// TIA Portal V19 export
FUNCTION "HambaFiller" : Void   // FC100, STL
TITLE = Hamba Filler
{ S7_Optimized_Access := 'TRUE' }
VERSION : 0.0
// Comment
// stored: AutoNumber false
BEGIN

NETWORK
TITLE = CIP of Transfer line
      CLR;

      A     "CIP_Hamba_bit_00";
      JC    M015;

      A     "CIP_Hamba_bit_02";  // If system is requested to stop
      AN    "CIP_Route_Request";  // by loss of Route request
      JC    M015;  // It does a controlled shutdown

      A     "CIP_Hamba_bit_02";  // Once CIP Route is started it continues
      JC    M002;  // Unless the Route request is lost


      A     "CIP_Route_Request";
      AN    "Product_Request";
      AN    "Steam_Request";
      A     "CIP Stop Push Button";
      AN    "RTE_404_DB".HMI.RUNNING;
      JCN   M001;

      S     "CIP_Hamba_bit_02";
M002: R     "MY0902";  //turn off steam supply
      R     "MY0909";  //turn off steam to barrier
      A     "CIP_Hamba_bit_03";  //Once Y0909R is proved stop checking
      JC    M016;

      A     "Y0909R";  //check valve de-energised
      A     "PG_Devices".DI_100_005_X06_X1_3p2;  // Polygon Filler transfer line blanked off
      JCN   M001;

      S     "CIP_Hamba_bit_03";
M016: S     "MY0908";  //open 'product' route
      S     "MY0910";  //open 'product' route

      A     "Y0908S";  //check valve energised
      A     "Y0910S";  //check valve energised
      JCN   M001;

      S     "M_Cip_Route";
      S     "CIP_Hamba_bit_00";
      JU    M001;

// Start of Loss of CIP Route Request shutdown sequence
M015: CLR;
      A     "CIP_Hamba_bit_01";  //Awaiting CIP Drain Timer End
      JC    M013;

      A     "CIP_Route_Request";
      A     "CIP Stop Push Button";
      S     "M_Cip_Route";  //CORRECT?

      A     "CIP_Route_Request";
      AN    "CIP_Hamba_bit_04";  // Once Shutdown has started
      JC    M001;  // It continues until completed

      S     "CIP_Hamba_bit_04";
      R     "MY0910";
      R     "M_Cip_Route";
      A     "CIP_Hamba_bit_05";  //Once Y0910R is proved stop checking
      JC    M014;

      A     "Y0910R";  //check valve de-energised
      JCN   M001;

      S     "CIP_Hamba_bit_05";
M014: S     "MY0911";
      A     "Y0911S";  //check valve energised
      JCN   M001;

      S     "TIM57";  // DrainingHambaTime
      S     "CIP_Hamba_bit_01";
      JU    M001;

M013: CLR;
      A     "Tag_69";
      JC    M001;
      R     "MY0911";
      R     "MY0908";
      R     "CIP_Hamba_bit_00";
      R     "CIP_Hamba_bit_01";
      R     "CIP_Hamba_bit_02";
      R     "CIP_Hamba_bit_03";
      R     "CIP_Hamba_bit_04";
      R     "CIP_Hamba_bit_05";

M001: CLR;
      A     "CIP_Running";
      =     "MX0913";  //set cip running bit

      A     "M_Cip_Route";  //cip route is active
      A(;
      O     "ItemAlarmsOP".Item[20];  //FB_FAULT_VALVE_09_05
      O     "ItemAlarmsOP".Item[23];  //FB_FAULT_VALVE_09_08
      O     "ItemAlarmsOP".Item[24];  //FB_FAULT_VALVE_09_09
      O     "ItemAlarmsOP".Item[25];  //FB_FAULT_VALVE_09_10
      O     "ItemAlarmsOP".Item[26];  //FB_FAULT_VALVE_09_11
      ON    "PG_Devices".DI_100_005_X06_X1_3p2;  // Polygon Filler transfer line blanked off
      );
      R     "M_Cip_Route";  //reset cip route active flag if valve in fault

NETWORK
TITLE = CIp Stop Push Button Operated Alarm and Stop CIP route signal
      AN    "CIP Stop Push Button";
      S     "ProcessAndPbAlarms"."A"[63];  //A63_Stop_CIP_PB_Operated
      R     "M_Cip_Route";

NETWORK
TITLE = SIP of Transfer line
      A     "steam_lp_request";  // If LP steam is requested
      R     "MY0903";  //
      S     "MY0902";

      A     "steam_lp_request";  // If LP steam is requested
      AN    "MY0903";  // if Y0903 is being asked to close
      A     "MY0902";  // and Y0902 is being asked to open
      =     "M_LP_Steam_ON";  // then, inform that the LP steam request has been actioned


      CLR;

      A     "SIP_Hamba_bit_00";
      JC    M005;

      A     "SIP_Hamba_bit_02";  // If system is requested to stop
      A(;  // After it has been started
      ON    "Steam_Request";  // It does a controlled shutdown
      ON    "Barrier_Sterile";
      );
      S     "SIP_Hamba_bit_00";
      JC    M005;

      A     "Steam_Request";
      A     "Barrier_Sterile";
      JCN   M004;

      S     "SIP_Hamba_bit_02";
      R     "MY0902";
      R     "MY0910";
      R     "MY0911";
      A     "SIP_Hamba_bit_04";  //Once Y0910R and Y0911R are proved
      JC    M003;  //Stop checking

      A     "Y0910R";  //check valve de-energised
      A     "Y0911R";  //check valve de-energised
      JCN   M004;

      S     "SIP_Hamba_bit_04";
M003: S     "MY0908";
      S     "MY0909";
      A     "Y0908S";  //check valve energised
      A     "Y0909S";  //check valve energised
      JCN   M004;

      S     "MY0903";
      S     "M_Sip_Steam";
      S     "SIP_Hamba_High_SteamPres";
      R     "SIP_Hamba_Low_SteamPres";
      S     "SIP_Hamba_bit_00";
      JU    M004;

// Start of Loss of SIP Route Request shutdown sequence
M005: CLR;
      A     "SIP_Hamba_bit_01";
      JC    M017;

      A     "Steam_Request";
      AN    "SIP_Hamba_bit_03";
      JC    M004;

      S     "SIP_Hamba_bit_03";
      R     "MY0908";
      R     "SIP_Hamba_High_SteamPres";
      A     "Y0908R";  //check valve de-energised
      JCN   M004;

      R     "M_Sip_Steam";
      R     "MY0903";
      S     "MY0902";
      S     "SIP_Hamba_Low_SteamPres";
      S     "SIP_Hamba_bit_01";
      JC    M004;

M017: CLR;
      A     "ATI";
      R     "SIP_Hamba_bit_00";
      R     "SIP_Hamba_bit_01";
      R     "SIP_Hamba_bit_02";
      R     "SIP_Hamba_bit_03";
      R     "SIP_Hamba_bit_04";
      R     "SIP_Hamba_bit_05";

M004: NOP   0;

      AN    "Barrier_Sterile";
      R     "SIP_Hamba_High_SteamPres";
      R     "SIP_Hamba_Low_SteamPres";
      CLR;

      A(;
      O     "ItemAlarmsOP".Item[23];  //FB_FAULT_VALVE_09_08
      O     "ItemAlarmsOP".Item[24];  //FB_FAULT_VALVE_09_09
      O     "ItemAlarmsOP".Item[25];  //FB_FAULT_VALVE_09_10
      O     "ItemAlarmsOP".Item[26];  //FB_FAULT_VALVE_09_11
      O     "steam_lp_request";  // If LP steam is requested
      );
      R     "M_Sip_Steam";
      CLR;

      AN    "ItemAlarmsOP".Item[23];  //FB_FAULT_VALVE_09_08
      AN    "ItemAlarmsOP".Item[24];  //FB_FAULT_VALVE_09_09
      AN    "ItemAlarmsOP".Item[25];  //FB_FAULT_VALVE_09_10
      AN    "ItemAlarmsOP".Item[26];  //FB_FAULT_VALVE_09_11
      A     "MY0903";
      S     "M_Sip_Steam";
      CLR;

      AN    "TANK STERILE";
      R     "M_Barrier_Sterile";
      CLR;
      A     "Y0119S";
      R     "MY0902";
      R     "MY0903";
      R     "MY0909";
      R     "SIP_Hamba_Low_SteamPres";

NETWORK
TITLE = SIP of Transfer line Temp. check/alarm high
      A     "MY0903";
      A(;
      L     "MeasuredValues".TT0950REAL;
      L     "Setpoints_Hamba".TT0950BarrierTempHigh;
      <R;
      );
      L     "TIMER DATA BLOCK".SETPOINT_TIMER_58;
      SD    "Tag_99";
      NOP   0;
      NOP   0;
      NOP   0;
      A     "Tag_99";
      S     "ProcessAndPbAlarms"."A"[59];  //A59_TT0950TooLow
      R     "M_Sip_Steam";

NETWORK
TITLE = SIP of Transfer line Temp. check/alarm low
      A     "MY0902";
      A(;
      L     "MeasuredValues".TT0950REAL;
      L     "Setpoints_Hamba".TT0950BarrierTempLow;
      <R;
      );
      L     "TIMER DATA BLOCK".SETPOINT_TIMER_59;
      SD    "Tag_100";
      NOP   0;
      NOP   0;
      NOP   0;
      A     "Tag_100";
      S     "ProcessAndPbAlarms"."A"[60];  //A60_TT0950Low

NETWORK
TITLE = Product Routing
// ; Product available
      A     "M_PROD_AVAILABLE";
      FP    "One_shut_on";
      S     "M_Product_Available";

      AN    "M_PROD_AVAILABLE";
      FP    "One_shut_off";
      R     "M_Product_Available";

//; Product Routing

      A     "Prod_Hamba_bit_00";
      JC    M006;

      A     "Prod_Hamba_bit_08";  //If Product Route request
      AN    "Product_Request";  //Started but not complete
      S     "Prod_Hamba_bit_00";  //When Product request lost
      JC    M006;  //Go to Prod Route Shutdown

      A     "Product_Request";
      A     "MY0902";  //Cross check. V0902 will be energised if route selected.
      JCN   M007;
      S     "Prod_Hamba_bit_08";
      R     "MY0906";
      R     "MY0907";
      R     "MY0912";

      A     "Prod_Hamba_bit_09";  //Jump if Y0906R, Y0907R
      JC    M012;  //& Y0912R have been proved

      A     "Y0906R";  //check valve de-energised
      A     "Y0907R";  //check valve de-energised
      A     "Y0912R";  //check valve de-energised
      A     "Y0908R";  //check valve de-energised, closed on loss of "Steam_Request" Network 3
      JCN   M007;

      S     "Prod_Hamba_bit_09";
M012: S     "MY0904";
      S     "MY0905";
      A     "Y0904S";  //check valve energised
      A     "Y0905S";  //check valve energised
      JCN   M007;

      S     "M_Product_Route";
      S     "Prod_Hamba_bit_00";
      JU    M007;

//Start of loss of Product Route signal
M006: CLR;
      A     "Prod_Hamba_bit_01";
      JC    M00c;

      A     "Product_Request";  //Once Poduct route Shutdown
      AN    "Prod_Hamba_bit_10";  //Started set to ensure finishes
      JC    M007;

      S     "Prod_Hamba_bit_10";
      R     "M_Product_Route";
      R     "MY0904";
      R     "MY0905";
      S     "DisableMonitoringTT0951";
      A     "Prod_Hamba_bit_11";  //Jump if Y0904R & Y0905R
      JC    M008;  //have been proved

      A     "Y0904R";  //check valve de-energised
      A     "Y0905R";  //check valve de-energised
      JCN   M007;

      S     "Prod_Hamba_bit_11";
M008: S     "MY0907";
      S     "MY0912";
      A     "Prod_Hamba_bit_12";  //Jump if Y0907S & Y0912S
      JC    M009;  //have been proved

      A     "Y0907S";  //check valve energised
      A     "Y0912S";  //check valve energised
      JCN   M007;

      S     "Prod_Hamba_bit_12";
M009: S     "MY0906";
      A     "Y0906S";  //check valve energised
      JCN   M007;

      S     "TIM63";  // Y0912PurgeBarrierTime
      S     "Prod_Hamba_bit_01";
      JU    M007;

M00c: CLR;
      A     "Prod_Hamba_bit_02";
      JC    M00d;

      A     "Tag_71";
      JC    M007;
      R     "MY0912";
      R     "DisableMonitoringTT0951";
      A     "Y0912R";  //check valve de-energised
      JCN   M007;

      S     "Prod_Hamba_bit_02";
      JU    M007;

M00d: CLR;
      A     "ATI";
      R     "Prod_Hamba_bit_00";
      R     "Prod_Hamba_bit_01";
      R     "Prod_Hamba_bit_02";
      R     "Prod_Hamba_bit_08";
      R     "Prod_Hamba_bit_09";
      R     "Prod_Hamba_bit_10";
      R     "Prod_Hamba_bit_11";
      R     "Prod_Hamba_bit_12";

M007: CLR;
      AN    "Product_Request";
      R     "Prod_Hamba_bit_03";
      R     "Prod_Hamba_bit_04";
      R     "Prod_Hamba_bit_05";
      R     "Prod_Hamba_bit_06";
      R     "ProcessAndPbAlarms"."A"[61];  //A61_Hamba_Valve_Fault
      R     "ProcessAndPbAlarms"."A"[62];  //A62_Hamba_Barrier_low
      BEC;

//; Valve FB-error

      A     "Prod_Hamba_bit_03";
      AN    "Prod_Hamba_bit_04";
      JC    M010;

      AN    "ItemAlarmsOP".Item[19];  //FB_FAULT_VALVE_09_04
      AN    "ItemAlarmsOP".Item[20];  //FB_FAULT_VALVE_09_05
      AN    "ItemAlarmsOP".Item[21];  //FB_FAULT_VALVE_09_06
      AN    "ItemAlarmsOP".Item[22];  //FB_FAULT_VALVE_09_07
      AN    "ItemAlarmsOP".Item[27];  //FB_FAULT_VALVE_09_12
      JC    M00a;

      A     "Prod_Hamba_bit_03";
      JC    M010;
      R     "M_Product_Route";
      R     "MY0904";
      R     "MY0905";
      S     "DisableMonitoringTT0951";
      A     "Y0904R";  //check valve de-energised
      A     "Y0905R";  //check valve de-energised
      JCN   M00b;

      S     "MY0907";
      S     "MY0912";
      S     "MY0906";
      S     "TIM64";  // Y0912PurgeBarrierTime
      S     "ProcessAndPbAlarms"."A"[61];  //A61_Hamba_Valve_Fault
      S     "Prod_Hamba_bit_03";
      JU    M00b;

M010: CLR;
      A     "Prod_Hamba_bit_04";
      JC    M011;

      A     "Tag_72";
      JC    M00b;
      R     "MY0912";
      R     "DisableMonitoringTT0951";
      S     "Prod_Hamba_bit_04";
      JU    M00b;

M011: CLR;
      JU    M00b;

M00a: CLR;
      R     "Prod_Hamba_bit_03";
      R     "Prod_Hamba_bit_04";

M00b: CLR;

//; Low temperature TT 09.51

      A     "Prod_Hamba_bit_05";
      AN    "Prod_Hamba_bit_06";
      JC    M019;

      AN    "ProcessAndPbAlarms"."A"[58];  //A58_TT0951Low
      JC    M00e;

      A     "Prod_Hamba_bit_05";
      JC    M019;
      R     "M_Product_Route";
      S     "StopFillers_UHT_Rec";
      R     "MY0904";
      R     "MY0905";
      S     "DisableMonitoringTT0951";
      A     "Y0904R";  //check valve de-energised
      A     "Y0905R";  //check valve de-energised
      JCN   M00f;

      S     "MY0907";
      S     "MY0912";
      A     "Y0907S";  //check valve energised
      A     "Y0912S";  //check valve energised
      JCN   M00f;

      S     "MY0906";
      A     "Y0906S";  //check valve energised
      JCN   M00f;

      S     "TIM65";  // Y0912PurgeBarrierTime
      S     "ProcessAndPbAlarms"."A"[62];  //A62_Hamba_Barrier_low
      S     "Prod_Hamba_bit_05";
      JU    M00f;

M019: CLR;
      A     "Prod_Hamba_bit_06";
      JC    M018;

      A     "Tag_73";
      JC    M00f;
      R     "MY0912";
//    R     "DisableMonitoringTT0951"
      S     "Prod_Hamba_bit_06";
      JU    M00f;

M018: CLR;
      JU    M00f;

M00e: CLR;
      R     "Prod_Hamba_bit_05";
      R     "Prod_Hamba_bit_06";

M00f: CLR;

END_FUNCTION
